PROGRAM MAIN
VAR
nCase : INT;


	

END_VAR



IF GVL_Safety.HWStart THEN
	GVL_Safety.Run  := TRUE;
	GVL_Safety.Start := TRUE;
END_IF

IF  NOT GVL_Safety.HWStop THEN
	GVL_Safety.Run  := FALSE;
	GVL_Safety.Start := FALSE;
END_IF
		
IF 	GVL_Safety.HWReset THEN
	GVL_Safety.Reset := TRUE;
ELSE
	GVL_Safety.Reset := FALSE;	
END_IF


IF gvl_safety.SaeftyOk THEN
	gvl_safety.HWSafetyOk := TRUE;
ELSE	
	gvl_safety.HWSafetyOk := FALSE;
END_IF

IF NOT gvl_safety.SafetyInRun THEN
	gvl_safety.HWerror := TRUE;
ELSE	
	gvl_safety.HWerror := FALSE;
END_IF

END_PROGRAM

(* stored: Version 1.1.0.1, ProductVersion 3.1.4024.12
   POU MAIN: Id {1b4dff48-5fc4-4640-872d-67c650f13b5e}, SpecialFunc None *)
